(* PLC project Counter (OSIE), Unknown Unnamed 1 *)
(* stored: creationDateTime 2021-05-14T14:33:11, modificationDateTime 2021-06-03T16:47:18 *)

FUNCTION_BLOCK CounterST
  VAR_INPUT
    Reset : BOOL;
  END_VAR
  VAR_OUTPUT
    Out1 : INT;
    Out0 : INT;
  END_VAR
  VAR
    Cnt1 : INT;
    Cnt0 : INT;
  END_VAR
  VAR_EXTERNAL
    ResetCounterValue : INT;
    Relay0Value : BOOL;
    Relay1Value : BOOL;
    Relay2Value : BOOL;
    Relay3Value : BOOL;
  END_VAR

            IF Reset THEN
  Cnt0 := ResetCounterValue;
  Cnt1 := ResetCounterValue;
  Reset := False;
ELSE
  Cnt0 := Cnt0 + 1;
  Cnt1 := Cnt1 + 1;
  IF Cnt1 > 10 THEN
    Relay0Value := True;
    Relay1Value := True;
  ELSE
    Relay0Value := True;
    Relay1Value := False;
  END_IF;
  
  IF Cnt1 > 15 THEN
    Relay1Value := False;
    Cnt1 :=0;
  END_IF;
  
END_IF;

Out1 := Cnt1;
Out0 := Cnt0;
          
END_FUNCTION_BLOCK

PROGRAM plc_prg
  VAR_INPUT
    Reset : BOOL;
  END_VAR
  VAR_OUTPUT
    Cnt0 : INT;
    Cnt1 : INT;
  END_VAR
  VAR
    CounterST0 : CounterST;
  END_VAR

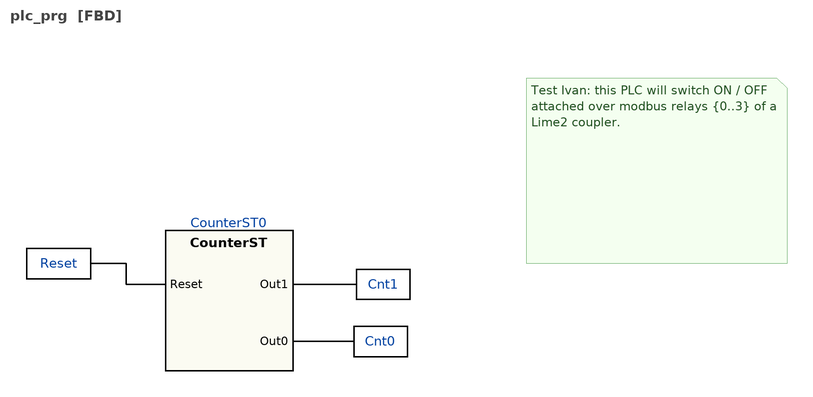
(* FBD diagram, written out as Structured Text *)
(* Test Ivan: this PLC will switch ON / OFF attached over modbus relays {0..3} of a Lime2 coupler. *)
CounterST0(Reset := Reset);
Cnt1 := CounterST0.Out1;
Cnt0 := CounterST0.Out0;
END_PROGRAM

CONFIGURATION config
  VAR_GLOBAL
    ResetCounterValue : INT := 0;
    Relay0Value AT %QX0.0.0.0 : BOOL := 0;  (* The status of the Lime's relay0 (read over modbus) *)
    Relay1Value AT %QX0.0.1.1 : BOOL := 0;  (* The status of the Lime's relay1 (read over modbus) *)
    Relay2Value AT %QX0.0.2.2 : BOOL := 0;  (* The status of the Lime's relay2 (read over modbus) *)
    Relay3Value AT %QX0.0.3.3 : BOOL := 0;  (* The status of the Lime's relay3 (read over modbus) *)
  END_VAR
  RESOURCE resource1 ON PLC
    TASK task0(INTERVAL := T#20ms, PRIORITY := 0);
    PROGRAM instance0 WITH task0 : plc_prg;
  END_RESOURCE
END_CONFIGURATION
